# EPICS substitutions: utcaApp/Db/user.substitutions
# Example substitutions file

file "db/dbExample1.db" {
    { user = "ericorolim" }
}

file db/dbExample2.db {
    pattern { user, no, scan }
        { "ericorolim", 1, "1 second" }
        { "ericorolim", 2, "2 second" }
        { "ericorolim", 3, "5 second" }
}
